FUNCTION_BLOCK E_DEMUX (* Event demultiplexer *)
  (* Standard: 61499-1; Classification: Event Processing; Function: Demultiplexing *)
  (* Version 0.1, 2002-01-29, JHC, Rockwell Automation, XML version *)
  (* Version 0.0, 1998-05-02, JHC, Rockwell Automation, SRC version *)
  (* Compiler header: package fb.rt.events; *)
  (* Compiler Java IBM VisualAge 3.0 *)
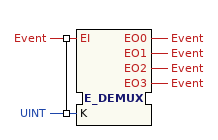
  EVENT_INPUT
    EI WITH K; (* Event to demultiplex *)
  END_EVENT
  EVENT_OUTPUT
    EO0;
    EO1;
    EO2;
    EO3; (* Number of outputs is implementation dependent *)
  END_EVENT
  VAR_INPUT
    K : UINT; (* Event index,maximum is implementation dependent *)
  END_VAR
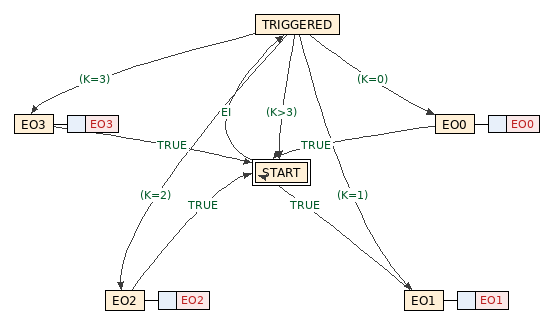
  EC_STATES
    START; (* Initial State *)
    TRIGGERED; (* Intermediate state after EI arrives *)
    EO0 : -> EO0;
    EO1 : -> EO1;
    EO2 : -> EO2;
    EO3 : -> EO3;
  END_STATES
  EC_TRANSITIONS
    START TO TRIGGERED := EI;
    TRIGGERED TO EO0 := (K=0);
    TRIGGERED TO EO1 := (K=1);
    TRIGGERED TO EO2 := (K=2);
    TRIGGERED TO EO3 := (K=3);
    TRIGGERED TO START := (K>3);
    EO0 TO START := TRUE;
    EO1 TO START := TRUE;
    EO2 TO START := TRUE;
    EO3 TO START := TRUE;
  END_TRANSITIONS
END_FUNCTION_BLOCK
